// Converts TcLog.LogLevels into Tc2_System.ADSLOG_MSGTYPEs.
{attribute 'hide'}
FUNCTION INTERNAL LogLevelToAdsLogMsgType : DWORD
VAR_INPUT
  logLevel : LogLevels;
END_VAR
VAR
  _retVal : DWORD;
END_VAR

CASE logLevel OF
  LogLevels.Debug, LogLevels.Information:
    _retVal := Tc2_System.ADSLOG_MSGTYPE_HINT;
  LogLevels.Warning:
    _retVal := Tc2_System.ADSLOG_MSGTYPE_WARN;
  LogLevels.Error, LogLevels.Fatal:
    _retVal := Tc2_System.ADSLOG_MSGTYPE_ERROR;
  ELSE
    _retVal := Tc2_System.ADSLOG_MSGTYPE_HINT;
END_CASE

LogLevelToAdsLogMsgType := _retVal;

END_FUNCTION

(* stored: Version 1.1.0.1, ProductVersion 3.1.4024.12
   POU LogLevelToAdsLogMsgType: Id {c5255ff0-b51b-42de-ab62-e7b30a9b316a}, SpecialFunc None *)
